// TIA Portal V18 export
// export: Created 2026-07-16T07:47:40.8959068Z, ExportSetting WithDefaults, DisplayName Totally Integrated Automation Portal, DisplayVersion V18 Update 5, DisplayName TIA Portal Openness, DisplayVersion V18 Update 5, DisplayName TIA Portal Version Control Interface, DisplayVersion V18, DisplayName SINAMICS Startdrive Advanced, DisplayVersion V18 SP2 Update 1, DisplayName SINAMICS Startdrive G110M, G120, G120C, G120D, G120P, G115D, DisplayVersion V18 SP2 Update 1, DisplayName SINAMICS Startdrive G130, G150, S120, S150, SINAMICS MV, S210, G220, S200, DisplayVersion V18 SP2 Update 1, DisplayName STEP 7 Professional, DisplayVersion V18 Update 5, DisplayName STEP 7 Safety, DisplayVersion V18, DisplayName WinCC Advanced / Unified PC, DisplayVersion V18 Update 5
FUNCTION "TEMPLATE--v1.1--04_ESTOP" : Void   // FC26, F_FBD
TITLE = SAFETY/EMERGENCY POWER CUT MANAGEMENT
{ S7_Optimized_Access := 'TRUE' }
VERSION : 0.1
// v1.0 First Emission
// V1.1 Generalized, Cumulatives now live in 02_COM
// stored: AutoNumber true, IsIECCheckEnabled false, UDAEnableTagReadback false
BEGIN

REGION Network 1: !!NetworkComment$$ Safety STOP
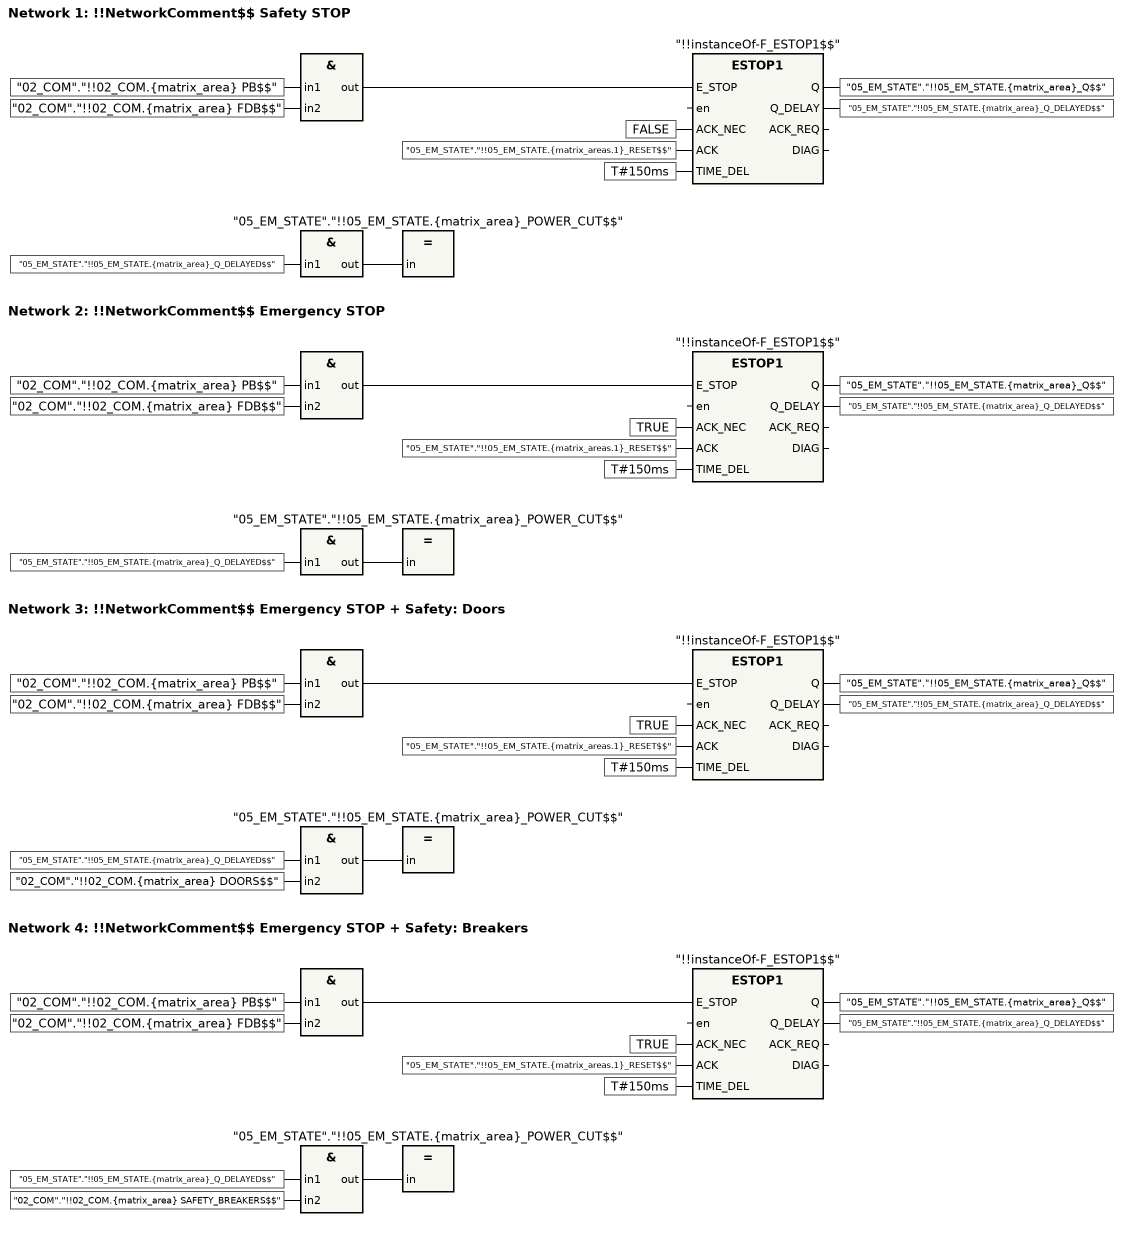
   "!!instanceOf-F_ESTOP1$$"(E_STOP := "02_COM"."!!02_COM.{matrix_area} PB$$" AND "02_COM"."!!02_COM.{matrix_area} FDB$$",   // ESTOP1
                           ACK_NEC := FALSE,
                           ACK := "05_EM_STATE"."!!05_EM_STATE.{matrix_areas.1}_RESET$$",
                           TIME_DEL := T#150ms,
                           Q => "05_EM_STATE"."!!05_EM_STATE.{matrix_area}_Q$$",
                           Q_DELAY => "05_EM_STATE"."!!05_EM_STATE.{matrix_area}_Q_DELAYED$$");
   "05_EM_STATE"."!!05_EM_STATE.{matrix_area}_POWER_CUT$$" := "05_EM_STATE"."!!05_EM_STATE.{matrix_area}_Q_DELAYED$$";
END_REGION

REGION Network 2: !!NetworkComment$$ Emergency STOP
   "!!instanceOf-F_ESTOP1$$"(E_STOP := "02_COM"."!!02_COM.{matrix_area} PB$$" AND "02_COM"."!!02_COM.{matrix_area} FDB$$",   // ESTOP1
                           ACK_NEC := TRUE,
                           ACK := "05_EM_STATE"."!!05_EM_STATE.{matrix_areas.1}_RESET$$",
                           TIME_DEL := T#150ms,
                           Q => "05_EM_STATE"."!!05_EM_STATE.{matrix_area}_Q$$",
                           Q_DELAY => "05_EM_STATE"."!!05_EM_STATE.{matrix_area}_Q_DELAYED$$");
   "05_EM_STATE"."!!05_EM_STATE.{matrix_area}_POWER_CUT$$" := "05_EM_STATE"."!!05_EM_STATE.{matrix_area}_Q_DELAYED$$";
END_REGION

REGION Network 3: !!NetworkComment$$ Emergency STOP + Safety: Doors
   "!!instanceOf-F_ESTOP1$$"(E_STOP := "02_COM"."!!02_COM.{matrix_area} PB$$" AND "02_COM"."!!02_COM.{matrix_area} FDB$$",   // ESTOP1
                           ACK_NEC := TRUE,
                           ACK := "05_EM_STATE"."!!05_EM_STATE.{matrix_areas.1}_RESET$$",
                           TIME_DEL := T#150ms,
                           Q => "05_EM_STATE"."!!05_EM_STATE.{matrix_area}_Q$$",
                           Q_DELAY => "05_EM_STATE"."!!05_EM_STATE.{matrix_area}_Q_DELAYED$$");
   "05_EM_STATE"."!!05_EM_STATE.{matrix_area}_POWER_CUT$$" := "05_EM_STATE"."!!05_EM_STATE.{matrix_area}_Q_DELAYED$$" AND "02_COM"."!!02_COM.{matrix_area} DOORS$$";
END_REGION

REGION Network 4: !!NetworkComment$$ Emergency STOP + Safety: Breakers
   "!!instanceOf-F_ESTOP1$$"(E_STOP := "02_COM"."!!02_COM.{matrix_area} PB$$" AND "02_COM"."!!02_COM.{matrix_area} FDB$$",   // ESTOP1
                           ACK_NEC := TRUE,
                           ACK := "05_EM_STATE"."!!05_EM_STATE.{matrix_areas.1}_RESET$$",
                           TIME_DEL := T#150ms,
                           Q => "05_EM_STATE"."!!05_EM_STATE.{matrix_area}_Q$$",
                           Q_DELAY => "05_EM_STATE"."!!05_EM_STATE.{matrix_area}_Q_DELAYED$$");
   "05_EM_STATE"."!!05_EM_STATE.{matrix_area}_POWER_CUT$$" := "05_EM_STATE"."!!05_EM_STATE.{matrix_area}_Q_DELAYED$$" AND "02_COM"."!!02_COM.{matrix_area} SAFETY_BREAKERS$$";
END_REGION

REGION Network 5: !!NetworkComment$$ Emergency STOP + Safety: Doors, Breakers
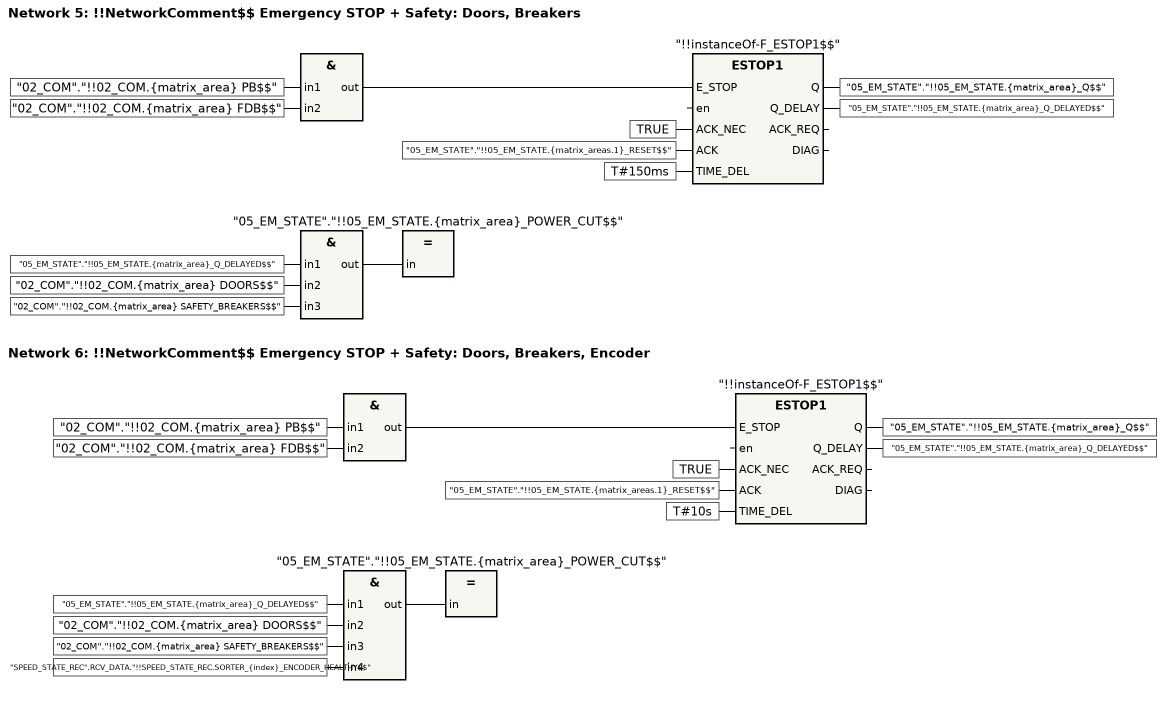
   "!!instanceOf-F_ESTOP1$$"(E_STOP := "02_COM"."!!02_COM.{matrix_area} PB$$" AND "02_COM"."!!02_COM.{matrix_area} FDB$$",   // ESTOP1
                           ACK_NEC := TRUE,
                           ACK := "05_EM_STATE"."!!05_EM_STATE.{matrix_areas.1}_RESET$$",
                           TIME_DEL := T#150ms,
                           Q => "05_EM_STATE"."!!05_EM_STATE.{matrix_area}_Q$$",
                           Q_DELAY => "05_EM_STATE"."!!05_EM_STATE.{matrix_area}_Q_DELAYED$$");
   "05_EM_STATE"."!!05_EM_STATE.{matrix_area}_POWER_CUT$$" := "05_EM_STATE"."!!05_EM_STATE.{matrix_area}_Q_DELAYED$$" AND "02_COM"."!!02_COM.{matrix_area} DOORS$$" AND "02_COM"."!!02_COM.{matrix_area} SAFETY_BREAKERS$$";
END_REGION

REGION Network 6: !!NetworkComment$$ Emergency STOP + Safety: Doors, Breakers, Encoder
   "!!instanceOf-F_ESTOP1$$"(E_STOP := "02_COM"."!!02_COM.{matrix_area} PB$$" AND "02_COM"."!!02_COM.{matrix_area} FDB$$",   // ESTOP1
                           ACK_NEC := TRUE,
                           ACK := "05_EM_STATE"."!!05_EM_STATE.{matrix_areas.1}_RESET$$",
                           TIME_DEL := T#10s,
                           Q => "05_EM_STATE"."!!05_EM_STATE.{matrix_area}_Q$$",
                           Q_DELAY => "05_EM_STATE"."!!05_EM_STATE.{matrix_area}_Q_DELAYED$$");
   "05_EM_STATE"."!!05_EM_STATE.{matrix_area}_POWER_CUT$$" := "05_EM_STATE"."!!05_EM_STATE.{matrix_area}_Q_DELAYED$$" AND "02_COM"."!!02_COM.{matrix_area} DOORS$$" AND "02_COM"."!!02_COM.{matrix_area} SAFETY_BREAKERS$$" AND "SPEED_STATE_REC".RCV_DATA."!!SPEED_STATE_REC.SORTER_{index}_ENCODER_HEALTHY$$";
END_REGION
END_FUNCTION
